RoboDK station: Estacion_feria_Con_Emergencia.rdk

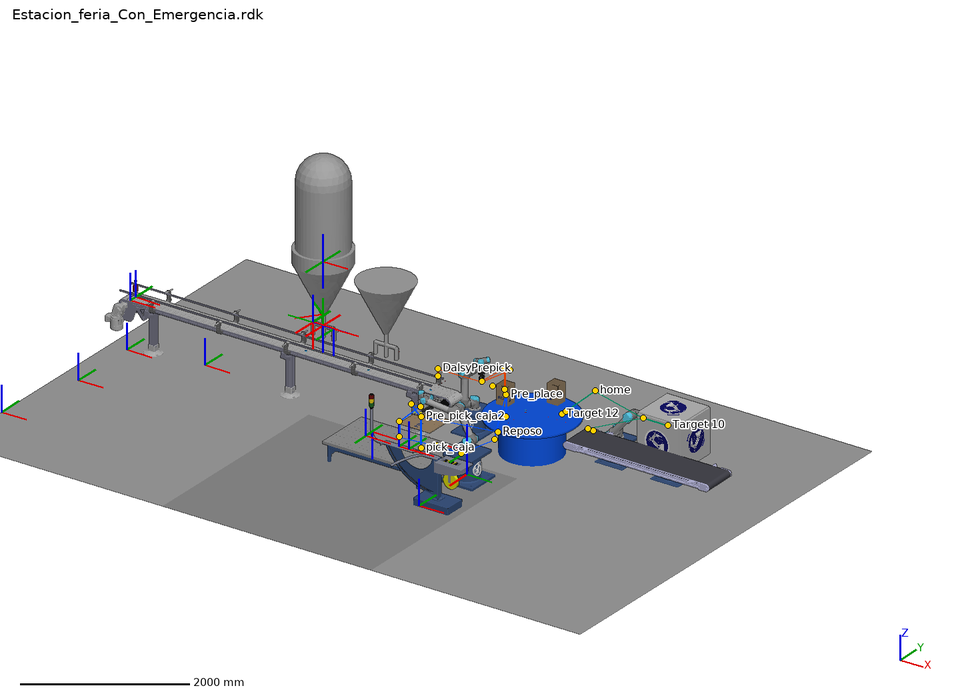
[picture v0: the station drawn from its stored meshes, robots at their saved joint values, targets as dots, program paths as lines]
Station EstacionProyectoFinaleliminarBotela (saved by RoboDK 5.9.4). Poses are relative to the parent item; angles as X-Y-Z fixed-axis rotations.
Station parameters (name, value as stored): Posicion, [[ 2850.000 ]] , CantBot1, 0, NUMBOTELLA1, 0, ElimBotellas1, 0, detectado1, 0, repes1, 0, Prellena1, 0, Prellena, 0, Detectado1, 0, IO_5, 1, NewPick, 0, Pinza, 1, NewPlace, 0, waituntil Detectado1, 1, Ventosa_plegado_caja, 1, CantCaja, 0.0, SCajaInicial, 0, SCajaPlace, 0, if(SCajaInicial, SyntaxError: Unexpected token `=', If(SCajaInicial, SyntaxError: Unexpected token `=', Mesa, 1, Mesa1, 0, Mesa2, 0, Mesa3, 1, MesaE, 1, MesaS, 1, Temperatura, 0, LotesPendientes, 1, SensorMqtt, 0, Ini_Detecta_Caja, 0, EMERGENCIA, 0
  - folder ESTACIÓN
    - folder Suelo
      - object Floor at (4500, 1500, 0) mm, size 3000 x 3000 x 0 mm, geometry from Floor.sld
      - object Floor2 at (1500, 1500, 0) mm, size 3000 x 3000 x 0 mm, geometry from Floor.sld
      - object Floor3 at (1500, 4500, 0) mm, size 3000 x 3000 x 0 mm, geometry from Floor.sld
      - object Floor4 at (4500, 4500, 0) mm, size 3000 x 3000 x 0 mm, geometry from Floor.sld
      - object Floor6 at (7500, 1500, 0) mm, size 3000 x 3000 x 0 mm, geometry from Floor.sld
      - object Floor5 at (7500, 4500, 0) mm, size 3000 x 3000 x 0 mm, geometry from Floor.sld
    - folder EMERGENCIA
      - program EMERGENCIA (3 instructions, listed below)
  - frame SisGeneral at (0, -19.13, 0) mm
    - folder SuministraCajas
      - frame SisCajas at (0, 1000, 0) mm
        - frame UR5 Base Cajas at (5520.28, 1665, 362.1) mm, rotated rx 0 ry 0 rz 180 deg
          - robot UR5 PrepCajas (model UR5): 6 axes
              modified DH rows (alpha deg, a mm, theta deg, d mm): 0, 0, 0, 89.2; 90, 0, 180, 0; 0, 425, 0, 0; 0, 392, 0, 109.3; -90, 0, 0, 94.75; 90, 0, 180, 82.5
              joint limits [-360, -360, -360, -360, -360, -360] to [360, 360, 360, 360, 360, 360]; home [0, -90, -90, 0, 90, 0]; saved at [7.72, -115.341, -54.372, -100.287, 90, 97.72]
            - frame Generic Box Erector Gripper Base at (0, 1000, 0) mm
            - robot Vplegadocaja: 1 axes
                modified DH rows (alpha deg, a mm, theta deg, d mm): 0, 0, 0, 0
                base shift (0, -125, 110) mm, rotated rx 0 ry 90 rz 0 deg
                joint limits [0] to [90]; home [0]; saved at [90]
              - tool Ventosa_plegado_caja, TCP at (0, 0, 200) mm
                - object Caja_plegada at (-6.06, -103.79, -200.38) mm, rotated rx 0 ry -90 rz 0 deg, size 213.4 x 213.4 x 444 mm, geometry from Box-215x215mm-Fold-2.sld
                - object caja_cintada at (15.94, -103.79, -200.38) mm, rotated rx 0 ry -90 rz 0 deg, size 160.1 x 160.1 x 259.7 mm, geometry from Box-215x215mm-Fold-3.sld
                - object Caja at (-171.32, 14.39, -556.39) mm, rotated rx 90 ry 0 rz 0 deg, size 444 x 419.7 x 11.5 mm, geometry from Box-215x215mm-Unfolded.sld
          - frame CoordBase_pedestal_caja at (-4.43, 0, -300) mm, rotated rx 0 ry 0 rz 90 deg
            - object Pedestal R1 at (0, 0, -60) mm, size 480 x 480 x 365.8 mm, geometry from Pedestal-H12in-Type-1.sld
          - target Reposo (Cartesian target) at (-498.67, 66.18, 420.87) mm, rotated rx 178.02 ry -0.17 rz 90 deg; joints [184.99, -90.98, -90.12, -90.89, 90, 4.99] of UR5 PrepCajas
          - target Pre_pick_caja2 (Cartesian target) at (671.03, -19.34, 260.81) mm, rotated rx 180 ry 0 rz 180 deg; joints [7.72, -117.384, -80.943, -71.673, 90, 97.72] of UR5 PrepCajas
          - target pick_caja (Cartesian target) at (671.03, -19.34, -150.19) mm, rotated rx 180 ry 0 rz 180 deg; joints [7.72, -132.159, -91.765, -46.076, 90, 97.72] of UR5 PrepCajas
          - target Giro (Cartesian target) at (580.93, 308.91, 583.09) mm, rotated rx 0 ry 90 rz 90 deg; joints [31.389, -172.181, 52.722, -60.541, 148.611, 90] of UR5 PrepCajas
          - target Paso_cintadora (Cartesian target) at (395, 385.89, 633.19) mm, rotated rx -45 ry 90 rz 45 deg; joints [50.203, -102.986, -71.875, -5.139, 129.797, 90] of UR5 PrepCajas
          - target Pre_abajo (Cartesian target) at (425, 775.89, 583.19) mm, rotated rx -45 ry 90 rz 45 deg; joints [58.921, -126.768, -44.607, -8.625, 121.079, 90] of UR5 PrepCajas
          - target abajo (Cartesian target) at (425, 775.89, 383.19) mm, rotated rx -45 ry 90 rz 45 deg; joints [58.921, -129.684, -69.347, 19.031, 121.079, 90] of UR5 PrepCajas
          - target fin_abajo (Cartesian target) at (-65, 715.89, 383.19) mm, rotated rx -45 ry 90 rz 45 deg; joints [112.972, -103.11, -110.097, 33.206, 67.028, 90] of UR5 PrepCajas
          - target cinta_abajo (Cartesian target) at (-425, 715.89, 383.19) mm, rotated rx -45 ry 90 rz 45 deg; joints [144.814, -123.817, -79.292, 23.109, 35.186, 90] of UR5 PrepCajas
          - target Paso_mesa (Cartesian target) at (-584.3, 268.15, 429.86) mm, rotated rx -90 ry 90 rz 90 deg; joints [162.957, -116.563, -83.461, 20.024, 107.043, 90] of UR5 PrepCajas
          - target Pre_place (Cartesian target) at (-128.1, -624.3, 529.86) mm, rotated rx 45 ry 90 rz -45 deg; joints [266.879, -85.143, -106.269, 11.412, 93.122, 90] of UR5 PrepCajas
          - target Place (Cartesian target) at (-128.1, -624.3, 241.86) mm, rotated rx 45 ry 90 rz -45 deg; joints [266.879, -110.903, -128.99, 59.893, 93.122, 90] of UR5 PrepCajas
        - frame Mesa at (4197.94, 1472.94, 273.52) mm
          - object mesa_caja at (0, 0, 0) mm, size 1420 x 820 x 800 mm, geometry from Table-1400x800x800mm.sld
          - frame Mesa_caja at (480, 0, 0) mm
          - object Sensor_caja_inicial at (650, -170, 0) mm, rotated rx 0 ry 0 rz 90 deg, size 683.3 x 45.2 x 12.5 mm, geometry from SICK-WL4S-Laser-Sensor.sld
        - frame Sistema_plegadora at (5470, 760, 0) mm
          - frame Caja_plegadora at (-210, 90, 650) mm
          - object Box Erector Station at (180, 120, 0) mm, rotated rx 0 ry 0 rz -90 deg, size 477.6 x 1402.8 x 1195.5 mm, geometry from Box-Erector-Station.sld
      - folder Programas_RDK
        - program Pick_place_caja (41 instructions, listed below)
        - program Main_sensor (11 instructions, listed below)
      - folder Programas_python
        - Python program ResetCaja (listed below)
        - Python program 2_caja (listed below)
        - Python program 3_caja (listed below)
        - Python program Abrir_Herramienta (listed below)
        - Python program Cerrar_heramienta (listed below)
        - Python program Copiar_caja_place (listed below)
        - Python program Inicializar_contador (listed below)
        - Python program Sensor_inicial (listed below)
        - Python program Sensor_place (listed below)
        - Python program QuitarCajasOcultas (listed below)
    - folder CintayRobot
      - frame SisRefPick at (250, 2217.22, 0) mm
        - frame Cinta Botellas 1 at (0, 1000, 0) mm
          - robot CintaUno: 1 axes
              modified DH rows (alpha deg, a mm, theta deg, d mm): 0, 0, 0, 0 linear
              base shift (0, 0, 0) mm, rotated rx 0 ry 90 rz 0 deg
              joint limits [0] to [4500]; home [0]; saved at [50]
            - frame FrameBotellaSave at (0, 0, 0) mm
              - object Guardado at (0, 0, 0) mm, size 71.4 x 71.4 x 225.2 mm, geometry from Bottle-Label.sld
            - frame Move at (0, 0, 0) mm
              - frame FrameBotella at (0, 100, 0) mm
                - object Guardado at (0, 0, 0) mm, size 71.4 x 71.4 x 225.2 mm, geometry from Bottle-Label.sld
                - object botella0.0 at (0, 0, 0) mm, size 71.4 x 71.4 x 225.2 mm, geometry from Bottle-Label.sld
          - target Inicio (Cartesian target) at (0, 100, 863) mm; joints [0] of CintaUno
          - target Final (Cartesian target) at (4325.5, 559.3, 913.95) mm, rotated rx -90 ry 0 rz 90 deg; joints [0, -90, -90, 0, 90, 0] of CintaUno
          - frame TANQUE 1 at (1750, -902.14, 647.6) mm
            - frame Cono at (1000, 1000, 1240) mm, rotated rx 180 ry 0 rz 0 deg
              - object Cone 500x500mm at (0, 0, 0) mm, size 746.2 x 750 x 750 mm, geometry from Cone-500x500mm.sld
            - frame Deposito at (1000, 1000, 1240) mm
              - object Deposito at (0, 0, 0) mm, size 750 x 750 x 1389.5 mm, geometry from Light-Off.sld
            - frame Frame 24 at (1000.71, 1000.6, 551.36) mm, rotated rx 180 ry 0 rz -124.91 deg
              - object Cylinder 50x150mm at (0, 0, 0) mm, size 50 x 50 x 150 mm, geometry from Cylinder-50x150mm.sld
            - frame Frame 25 at (1000.71, 1000.6, 401.36) mm, rotated rx -180 ry 0 rz -90 deg
              - object Cylinder 50x150mm at (0, 0, 0) mm, size 50 x 50 x 150 mm, geometry from Cylinder-50x150mm.sld
            - frame Frame 26 at (1000.71, 1000.6, 401.36) mm, rotated rx 90 ry 0 rz 90 deg
              - object Cylinder 50x150mm at (0, 0, 0) mm, size 50 x 50 x 150 mm, geometry from Cylinder-50x150mm.sld
            - frame Frame 27 at (1150.71, 1000.6, 401.36) mm, rotated rx -180 ry 0 rz 0 deg
              - object Cylinder 50x150mm at (0, 0, 0) mm, size 50 x 50 x 150 mm, geometry from Cylinder-50x150mm.sld
            - frame Frame 25 at (1000.71, 1000.6, 401.36) mm, rotated rx -180 ry 0 rz -90 deg
              - object Cylinder 50x150mm at (0, 0, 0) mm, size 50 x 50 x 150 mm, geometry from Cylinder-50x150mm.sld
            - frame Frame 25 at (850.71, 1000.6, 401.36) mm, rotated rx -180 ry 0 rz -90 deg
              - object Cylinder 50x150mm at (0, 0, 0) mm, size 50 x 50 x 150 mm, geometry from Cylinder-50x150mm.sld
            - frame Frame 25 at (850.71, 1000.6, 401.36) mm, rotated rx 0 ry 90 rz 0 deg
              - object Cylinder 50x150mm at (0, 0, 0) mm, size 50 x 50 x 150 mm, geometry from Cylinder-50x150mm.sld
            - frame Frame 31 at (850.65, 1001.38, 406.13) mm
              - object Sphere D100mm at (0, 0, 0) mm, size 50 x 50 x 50 mm, geometry from Sphere-D100mm.sld
            - frame Frame 31 at (1151.57, 999.51, 402.52) mm
              - object Sphere D100mm at (0, 0, 0) mm, size 50 x 50 x 50 mm, geometry from Sphere-D100mm.sld
          - frame DispensaTapones at (2650, -902.14, 647.6) mm
            - frame Cono at (1000, 1000, 1240) mm, rotated rx 180 ry 0 rz 0 deg
              - object Cone 500x500mm at (0, 0, 0) mm, size 746.2 x 750 x 750 mm, geometry from Cone-500x500mm.sld
            - frame Frame 24 at (1000.71, 1000.6, 551.36) mm, rotated rx 180 ry 0 rz -124.91 deg
              - object Cylinder 50x150mm at (0, 0, 0) mm, size 50 x 50 x 150 mm, geometry from Cylinder-50x150mm.sld
            - frame Frame 25 at (1000.71, 1000.6, 401.36) mm, rotated rx -180 ry 0 rz -90 deg
              - object Cylinder 50x150mm at (0, 0, 0) mm, size 50 x 50 x 150 mm, geometry from Cylinder-50x150mm.sld
            - frame Frame 26 at (1000.71, 1000.6, 401.36) mm, rotated rx 90 ry 0 rz 90 deg
              - object Cylinder 50x150mm at (0, 0, 0) mm, size 50 x 50 x 150 mm, geometry from Cylinder-50x150mm.sld
            - frame Frame 27 at (1150.71, 1000.6, 401.36) mm, rotated rx -180 ry 0 rz 0 deg
              - object Cylinder 50x150mm at (0, 0, 0) mm, size 50 x 50 x 150 mm, geometry from Cylinder-50x150mm.sld
            - frame Frame 25 at (1000.71, 1000.6, 401.36) mm, rotated rx -180 ry 0 rz -90 deg
              - object Cylinder 50x150mm at (0, 0, 0) mm, size 50 x 50 x 150 mm, geometry from Cylinder-50x150mm.sld
            - frame Frame 25 at (850.71, 1000.6, 401.36) mm, rotated rx -180 ry 0 rz -90 deg
              - object Cylinder 50x150mm at (0, 0, 0) mm, size 50 x 50 x 150 mm, geometry from Cylinder-50x150mm.sld
            - frame Frame 25 at (850.71, 1000.6, 401.36) mm, rotated rx 0 ry 90 rz 0 deg
              - object Cylinder 50x150mm at (0, 0, 0) mm, size 50 x 50 x 150 mm, geometry from Cylinder-50x150mm.sld
            - frame Frame 31 at (850.65, 1001.38, 406.13) mm
              - object Sphere D100mm at (0, 0, 0) mm, size 50 x 50 x 50 mm, geometry from Sphere-D100mm.sld
            - frame Frame 31 at (1151.57, 999.51, 402.52) mm
              - object Sphere D100mm at (0, 0, 0) mm, size 50 x 50 x 50 mm, geometry from Sphere-D100mm.sld
          - frame Sensor3 at (3498.8, -14.22, 715.35) mm, rotated rx 0 ry 0 rz 88.62 deg
            - object B2 at (0, 0, 0) mm, size 683.3 x 45.2 x 12.5 mm, geometry from SICK-WL4S-Laser-Sensor.sld
          - frame Sensor2 at (4402.28, -29.98, 715.35) mm, rotated rx 0 ry 0 rz 88.62 deg
            - object B1 at (0, 0, 0) mm, size 683.3 x 45.2 x 12.5 mm, geometry from SICK-WL4S-Laser-Sensor.sld
          - frame Sensor1 at (2598.8, -14.22, 715.35) mm, rotated rx 0 ry 0 rz 88.62 deg
            - object B0 at (0, 0, 0) mm, size 683.3 x 45.2 x 12.5 mm, geometry from SICK-WL4S-Laser-Sensor.sld
          - target DalsyPrepick (Cartesian target) at (4404.64, 97.25, 945.23) mm, rotated rx -179.46 ry -0.56 rz 92.6 deg; joints [67.794, -102.103, -28.32, -139.861, 89.279, 65.196] of UR5PickDalsy
          - target DalsyPick (Cartesian target) at (4400.29, 94.49, 846.14) mm, rotated rx -179.46 ry -0.56 rz 92.6 deg; joints [67.407, -90.716, -60.305, -119.258, 89.278, 64.809] of UR5PickDalsy
          - target DalsyPuntoPaso (Cartesian target) at (4989.54, 154.84, 921.17) mm, rotated rx 176.54 ry 3.78 rz 107.72 deg; joints [150.48, -91.95, -47.39, -125.54, 89.98, 132.65] of UR5PickDalsy
          - target PuntoDePaso2 (Cartesian target) at (5091.93, 592.06, 921.34) mm, rotated rx 176.53 ry 3.81 rz 169.24 deg; joints [212.01, -91.94, -47.38, -125.53, 89.97, 132.65] of UR5PickDalsy
          - target PrePlace (Cartesian target) at (5051.88, 544.46, 950.34) mm, rotated rx 179.87 ry 0 rz -95.46 deg; joints [208.979, -92.535, -38.825, -138.744, 90.075, 34.439] of UR5PickDalsy
          - target DalsyPlace (Cartesian target) at (5051.88, 544.46, 680.34) mm, rotated rx 179.87 ry 0 rz -95.46 deg; joints [208.979, -74.687, -99.618, -95.799, 90.075, 34.439] of UR5PickDalsy
          - target Target 9 (Cartesian target) at (5079.28, 251.73, 846.24) mm, rotated rx -179.45 ry -0.55 rz -167.69 deg; joints [167.11, -90.71, -60.3, -119.25, 89.27, 64.8] of UR5PickDalsy
          - target Target 10 (Cartesian target) at (7103.35, 957.35, 614.14) mm, rotated rx -138.15 ry 89.07 rz -48.26 deg; joints [177.195, -131.024, -49.86, -164.778, 177.217, -76.295] of UR5 SalidaCjas
          - target Target 11 (Cartesian target) at (4404.64, 97.25, 945.23) mm, rotated rx -179.46 ry -0.56 rz 92.6 deg; joints [67.794, -102.103, -28.32, -139.861, 89.279, 65.196] of UR5PickDalsy
          - target Target 12 (Cartesian target) at (5875.13, 535.29, 591.77) mm, rotated rx -124.69 ry 88.93 rz 144.57 deg; joints [23.154, -118.729, -72.709, -170.068, 203.904, -92.258] of UR5 SalidaCjas
        - frame UR5 BasePickDalsy at (4673.46, 1459.5, 355) mm, rotated rx 0 ry 0 rz 180 deg
          - robot UR5PickDalsy (model UR5): 6 axes
              modified DH rows (alpha deg, a mm, theta deg, d mm): 0, 0, 0, 89.2; 90, 0, 180, 0; 0, 425, 0, 0; 0, 392, 0, 109.3; -90, 0, 0, 94.75; 90, 0, 180, 82.5
              joint limits [-360, -360, -360, -360, -360, -360] to [360, 360, 360, 360, 360, 360]; home [0, -90, -90, 0, 90, 0]; saved at [150.48, -91.95, -47.39, -125.54, 89.98, 132.65]
            - tool GripperPick, TCP at (0, 0, 130) mm, size 147.4 x 75 x 146.8 mm
            - tool GripperPickV, TCP at (0, 0, 130) mm, size 134.4 x 75 x 157.6 mm
          - frame Frame 45 at (4.13, 0, -300) mm
            - object Pedestal R1 at (0, 0, 0) mm, size 400 x 400 x 304.8 mm, geometry from Pedestal-H12in-Type-1.sld
      - folder ProgramasDeLaCinta
        - Python program AvanzaCinta1 (listed below)
        - Python program AvanzaCinta2 (listed below)
        - Python program ResetBot (listed below)
        - program ProgCinta1 (15 instructions, listed below)
        - Python program ProgCintaUno (listed below)
      - folder Sensores
        - Python program ProgB0 (listed below)
        - Python program ProgB1 (listed below)
        - Python program ProgB2 (listed below)
      - folder ProgramasUr
        - program DalsyPickPlace (33 instructions, listed below)
        - Python program PickDalsy (listed below)
        - Python program PlaceDalsy (listed below)
        - Python program BorrarBotella (listed below)
        - Python program RobotPickAndPlace (listed below)
    - folder CerradoCajas
      - frame SisSalida at (6887.77, 2000, 0) mm
        - frame UR5BaseSalidaCajas at (-200.53, 2100.2, 305) mm, rotated rx 0 ry 0 rz 180 deg
          - robot UR5 SalidaCjas (model UR5): 6 axes
              modified DH rows (alpha deg, a mm, theta deg, d mm): 0, 0, 0, 89.2; 90, 0, 180, 0; 0, 425, 0, 0; 0, 392, 0, 109.3; -90, 0, 0, 94.75; 90, 0, 180, 82.5
              joint limits [-360, -360, -360, -360, -360, -360] to [360, 360, 360, 360, 360, 360]; home [0, -90, -90, 0, 90, 0]; saved at [177.195, -131.024, -49.86, -164.778, 177.217, -76.295]
            - tool VentosaSalida, TCP at (0, 22.5, 135) mm, size 179.2 x 110.2 x 138.7 mm
              - object caja_cerradaPLANTILLA at (2.18, 97.23, 6.23) mm, rotated rx 90.61 ry -0.74 rz -89.13 deg, size 160.1 x 160.1 x 186.3 mm, geometry from Box-215x215mm-Folded(2).sld
          - frame CoordBase at (0, 0, -320) mm, rotated rx -0.35 ry 0 rz 0 deg
            - object Pedestal R1 at (0, 0, 0) mm, size 400 x 400 x 304.8 mm, geometry from Pedestal-H12in-Type-1.sld
          - target pick_cajamesa (Cartesian target) at (562.11, 347.69, 286.77) mm, rotated rx -124.69 ry 88.93 rz -35.43 deg; joints [23.154, -118.729, -72.709, -170.068, 203.904, -92.258] of UR5 SalidaCjas
          - target prepick_cajamesa (Cartesian target) at (561.01, 262.7, 287.67) mm, rotated rx -124.69 ry 88.93 rz -35.43 deg; joints [15.242, -116.952, -75.276, -169.987, 195.996, -93.011] of UR5 SalidaCjas
          - target home (Cartesian target) at (209.75, 166.03, 613.52) mm, rotated rx -26.26 ry 79.18 rz 65.79 deg; joints [15.24, -64.23, -88.13, -169.98, 195.99, -58.26] of UR5 SalidaCjas
          - frame SisCubo at (-800, 0, -320) mm, rotated rx -0.35 ry 0 rz 0 deg
            - object Pedestal R1 at (0, 0, 0) mm, size 400 x 400 x 304.8 mm, geometry from Pedestal-H12in-Type-1.sld
            - object Cubo at (-300, -300, 300) mm, rotated rx 90 ry 0 rz 0 deg, size 636 x 636 x 672 mm
          - target pre_cajacubo (Cartesian target) at (-316.13, -74.99, 305.37) mm, rotated rx -138.15 ry 89.07 rz 131.74 deg; joints [174.473, -84.902, -111.44, -156.399, 174.538, -83.391] of UR5 SalidaCjas
          - target dentro_cajacubo (Cartesian target) at (-666.11, -74.37, 309.14) mm, rotated rx -138.15 ry 89.07 rz 131.74 deg; joints [177.195, -131.024, -49.86, -164.778, 177.217, -76.295] of UR5 SalidaCjas
          - target place_cajacinta (Cartesian target) at (-20.88, 535.48, 307.78) mm, rotated rx -142.74 ry 89.07 rz 36.86 deg; joints [81.199, -115.849, -73.914, 194.832, 171.57, 274.45] of UR5 SalidaCjas
          - target preplace_cajacinta (Cartesian target) at (54.12, 534.95, 308.76) mm, rotated rx -142.74 ry 89.07 rz 36.86 deg; joints [74.123, -120.474, -66.715, 189.969, 164.509, 272.115] of UR5 SalidaCjas
        - frame cinta2 at (-383.81, 1308.32, 516.62) mm, rotated rx 0.97 ry 0 rz 0 deg
          - robot CintaSalidas: 1 axes
              modified DH rows (alpha deg, a mm, theta deg, d mm): 0, 0, 0, 0 linear
              base shift (0, 0, 0) mm, rotated rx 0 ry 90 rz 0 deg
              joint limits [-500000] to [500000]; home [0]; saved at [-500000]
      - folder scripts
        - program Prog_cajasSalida (23 instructions, listed below)
        - folder pyt
          - Python program SensorDetectaCaja (listed below)
          - Python program Plantilla (listed below)
          - Python program AvanzaCajasSalida (listed below)
        - folder rdk
    - folder Mesa
      - frame MesaGiratoriaBase at (5724.13, 3717.02, 0) mm
        - robot MesaGiratoria: 1 axes
            modified DH rows (alpha deg, a mm, theta deg, d mm): 0, 0, 0, 0
            joint limits [-200] to [200]; home [0]; saved at [110]
          - frame SistMesaGiratoria at (0, 1000, 0) mm
          - frame Place_caja at (-410, 300, 573) mm, rotated rx 0 ry 0 rz -40 deg
            - object cajaplace1.0 at (310.2, 492.2, 15.02) mm, rotated rx 0 ry 0 rz -70 deg, size 160.1 x 160.1 x 259.7 mm, geometry from Box-215x215mm-Fold-3.sld
            - object cajaplace0.0 at (965.38, 230.44, 15.02) mm, rotated rx 0 ry 0 rz -160 deg, size 160.1 x 160.1 x 259.7 mm, geometry from Box-215x215mm-Fold-3.sld
        - folder ScriptsMesa
          - Python program MoverMesa (listed below)
          - program MoverMesaBucle (8 instructions, listed below)
        - object Sensor_place_caja at (-90, -30, 510) mm, rotated rx 0 ry 0 rz -90 deg, size 683.3 x 45.2 x 12.5 mm, geometry from SICK-WL4S-Laser-Sensor.sld
        - object SensorDetectaCajaSalida at (-100, -10, 510) mm, size 683.3 x 45.2 x 12.5 mm, geometry from SICK-WL4S-Laser-Sensor.sld
  - folder PROGRAMA_PRINCIPAL
    - program Main (17 instructions, listed below)
  - folder MQTT
    - Python program mqttlistenerCinta (listed below)
    - Python program RobotControllerCinta (listed below)
    - Python program mqttlistenerTEMP (listed below)
    - Python program mqttlistenerDecCaja (listed below)
    - Python program RobotControllerTEMP (listed below)
    - Python program RobotControllerDecCaja (listed below)
  - folder Basedatos
    - folder BaseDeDatos
      - Python program ConsultarBD (listed below)
      - Python program CrearBotellaBD (listed below)
      - Python program LlenarBD (listed below)
      - Python program ResetBD (listed below)
      - Python program EmpaquetarBD (listed below)
      - Python program TaponarBD (listed below)
    - folder JugarBD
      - Python program CrearLotesBD (listed below)
      - Python program TerminarLotesBD (listed below)
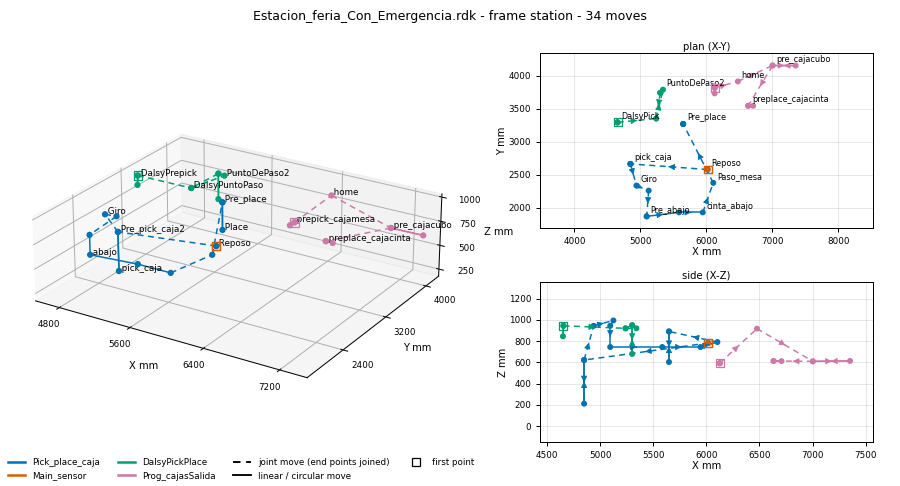
[picture p0: tool path of Estacion_feria_Con_Emergencia.rdk in frame station, 34 of 34 moves have a stored position in this frame; points joined in program order, loops and branches not executed]

--- program EMERGENCIA (robot UR5 PrepCajas) ---
  while EMERGENCIA ==1
  Pausa 500 ms
  end

--- program Pick_place_caja (robot UR5 PrepCajas) ---
  Est. Ref.: UR5 Base Cajas
  Est. herr: Ventosa_plegado_caja
  Establecer velocidad (500.0 mm/s)
  while Mesa==0
  Pausa 500 ms
  end
  Mesa=0
  MoveJ (Reposo)
  Llamar Abrir_Herramienta
  MoveJ (Pre_pick_caja2)
  Establecer velocidad (40.0 mm/s)
  MoveL (pick_caja)
  Set Ventosa_plegado_caja=1
  Adjuntar a Ventosa_plegado_caja
  Pausa 500 ms
  MoveL (Pre_pick_caja) -> target Pre_pick_caja2
  Establecer velocidad (500.0 mm/s)
  Llamar Cerrar_heramienta
  Llamar 2_caja
  Pausa 500 ms
  MoveJ (Giro)
  MoveJ (Paso_cintadora)
  MoveJ (Pre_abajo)
  Establecer velocidad (100.0 mm/s)
  MoveL (abajo)
  MoveL (fin_abajo)
  Llamar 3_caja
  MoveL (cinta_abajo)
  Establecer velocidad (500.0 mm/s)
  MoveJ (Paso_mesa)
  MoveJ (Pre_place)
  Establecer velocidad (100.0 mm/s)
  MoveL (Place)
  Set Ventosa_plegado_caja=0
  Separar de Ventosa_plegado_caja
  Pausa 500 ms
  Llamar Copiar_caja_place
  MoveL (Pre_place)
  Llamar ResetCaja
  Llamar QuitarCajasOcultas
  Mesa2=1

--- program Main_sensor (robot UR5 PrepCajas) ---
  Est. herr: Ventosa_plegado_caja
  Est. Ref.: UR5 Base Cajas
  MoveJ (Reposo)
  IF SCajaInicial == 1 THEN
  IF SCajaPlace==0 Then
  while Ini_Detecta_Caja == 0
  Pausa 500 ms
  end
  Llamar Pick_place_caja
  ENDIF
  ENDIF

--- Python program ResetCaja ---
from robodk import robolink
from robodk import robomath

# Conexión con RoboDK
RDK = robolink.Robolink()

# -------- OBTENER OBJETOS --------
caja = RDK.Item('Caja', robolink.ITEM_TYPE_OBJECT)
mesa_caja = RDK.Item('Mesa_caja', robolink.ITEM_TYPE_FRAME)

# -------- COMPROBACIONES --------
if not caja.Valid():
    raise Exception("No se encontró el objeto 'Caja'")

if not mesa_caja.Valid():
    raise Exception("No se encontró el sistema de coordenadas 'Mesa_caja'")

# -------- REINICIAR CAJA INICIAL --------

# Hacer que la caja dependa del frame Mesa_caja
caja.setParentStatic(mesa_caja)

# Definir la pose [x,y,z,rx,ry,rz] = [0,0,0,0,0,0] PARA PONERLO EN LA MESA
pose_origen = robomath.xyzrpw_2_pose([0, 0, 0, 0, 0, 0])

# Aplicar la pose a la caja
caja.setPose(pose_origen)

caja.setVisible(True,True)  #PONGO VISIBLE LA CAJA
RDK.Render()

#QUITO LAS CAJAS LAS CUALES USO PARA LA ANIMACION
caja2 = RDK.Item('Caja_plegada')
if not caja2.Valid():
    raise Exception('No se encontró el objeto Caja_plegada')

caja2.setVisible(False,False)
RDK.Render()

caja3=RDK.Item('Caja_cintada')
if not caja3.Valid():
    raise Exception('NO hay caja')

caja3.setVisible(False,False)
RDK.Render()

--- Python program 2_caja ---
# Type help("robodk.robolink") or help("robodk.robomath") for more information
# Press F5 to run the script
# Documentation: https://robodk.com/doc/en/RoboDK-API.html
# Reference:     https://robodk.com/doc/en/PythonAPI/robodk.html
# Note: It is not required to keep a copy of this file, your Python script is saved with your RDK project

# You can also use the new version of the API:
from robodk import robolink    # RoboDK API
from robodk import robomath    # Robot toolbox
RDK = robolink.Robolink()

from robodk.robolink import *
from robodk.robomath import *

#CODIGO DE LA CAJA SIN HACER NINGUNA MODIFICACION

cajainicial=RDK.Item('Caja') #CREO LA CAJA
if not cajainicial.Valid(): #COMPRUEBO QUE EXISTA LA CAJA
    raise Exception('Caja inicial no encontrada') #SINO LANZO UNA EXCEPCIONN

#------------------------------------------------
# CODIGGO PARA PONER CAJA '2ºESTADO' EN LA HERRAMIENTA

#HERRAMIENTA
tool = RDK.Item('Ventosa_plegado_caja', ITEM_TYPE_TOOL)#CREO ITEM HERRAMIENTA
if not tool.Valid(): #COMPRUEBO QUE EXISTA LA VENTOSA
    raise Exception('No se encontró la herramienta Ventosa_plegado_caja')#SINO LANZO UNA EXCEPCIONN
#----------------------------------------------------

#CAJA 2ºESTADO
caja = RDK.Item('Caja_plegada') #CREO LA CAJA EN SU 2ºESTADO
if not caja.Valid(): #COMPRUEBO QUE EXISTA ESA CAJA
    raise Exception('No se encontró el objeto Caja_plegada') #SINO LANZO UNA EXCEPCIONN

#----------------------------------------------------
# Hacer visible la caja
cajainicial.setVisible(False,False) #1.PONGO LA CAJA INICIAL INVISIBLE


#VOY A INSERTAR LA CAJA EN SU 2º ESTDO DENTRO DEL SISTEMA DE REFERENCIA DE LA VENTOSA
#ES DECIR PONDRE LA CAJA EN LA HERRAMIENTA POR CODIGO.
caja.setParentStatic(tool)

#VARIABLE POSE DONDE IRA LA CAJA
pose_herramienta = xyzrpw_2_pose([-6.063, -103.794, -200.377, 0, -90, 0])

# Aplicar la pose a la caja
caja.setPose(pose_herramienta)
# Hacer visible la caja
cajainicial.setVisible(False,False) #1.PONGO LA CAJA INICIAL INVISIBLE

caja.setVisible(True, True)

RDK.Render()

--- Python program 3_caja ---
# Type help("robodk.robolink") or help("robodk.robomath") for more information
# Press F5 to run the script
# Documentation: https://robodk.com/doc/en/RoboDK-API.html
# Reference:     https://robodk.com/doc/en/PythonAPI/robodk.html
# Note: It is not required to keep a copy of this file, your Python script is saved with your RDK project

# You can also use the new version of the API:
from robodk import robolink    # RoboDK API
from robodk import robomath    # Robot toolbox
RDK = robolink.Robolink()

from robodk.robolink import *
from robodk.robomath import *
#Fragmento de codigo donde hacemos invisible la caja sin cerrar la parte inferiro
caja=RDK.Item('Caja_plegada')
if not caja.Valid():
    raise Exception('No se encontro el objeto caja_plegada')

caja.setVisible(False,False)
RDK.Render()

#Fragmento de codigo donde hacemos invisible la caja con la parte inferior plegada
caja_abajo=RDK.Item('Caja_cintada')
tool=RDK.Item('Ventosa_plegado_caja', ITEM_TYPE_TOOL)
if not(caja_abajo.Valid()):
    raise Exception('Caja_cintada no se ha encontrado')
if not(tool.Valid()):
    raise Exception('No se ha conseguido unir a la ventosa')

caja_abajo.setVisible(True, True)
#Meter ne el sistema de referencia de la herramienta
caja_abajo.setParentStatic(tool)

pose_ventosa=xyzrpw_2_pose([15.937 , -103.794, -200.377, 0.00, -90.00, 0.00])
caja_abajo.setPose(pose_ventosa)
RDK.Render()

--- Python program Abrir_Herramienta ---
# Type help("robodk.robolink") or help("robodk.robomath") for more information
# Press F5 to run the script
# Documentation: https://robodk.com/doc/en/RoboDK-API.html
# Reference:     https://robodk.com/doc/en/PythonAPI/robodk.html
# Note: It is not required to keep a copy of this file, your Python script is saved with your RDK project

# You can also use the new version of the API:
from robodk import robolink    # RoboDK API
from robodk import robomath    # Robot toolbox

from robodk.robolink import Robolink

# Conectar con RoboDK
RDK = Robolink()

# Obtener la herramienta (mecanismo)
tool = RDK.Item('Vplegadocaja')

if not tool.Valid():
    raise Exception('No se encontró la herramienta Vplegadocaja')

# Obtener joints actuales de la herramienta
joints = tool.Joints().list()

if len(joints) == 0:
    raise Exception('La herramienta no tiene ejes articulares')

# Sumar 75 grados al eje deseado (J1 = índice 0)
joints[0] = joints[0] + 90

# Aplicar el pilotaje articular
tool.setJoints(joints)

--- Python program Cerrar_heramienta ---
# Type help("robodk.robolink") or help("robodk.robomath") for more information
# Press F5 to run the script
# Documentation: https://robodk.com/doc/en/RoboDK-API.html
# Reference:     https://robodk.com/doc/en/PythonAPI/robodk.html
# Note: It is not required to keep a copy of this file, your Python script is saved with your RDK project

# You can also use the new version of the API:
from robodk import robolink    # RoboDK API
from robodk import robomath    # Robot toolbox
RDK = robolink.Robolink()

from robodk.robolink import Robolink

import time

# Conectar con RoboDK
RDK = Robolink()

# Obtener la herramienta (mecanismo)
tool = RDK.Item('Vplegadocaja')

if not tool.Valid():
    raise Exception('No se encontró la herramienta Vplegadocaja')

# Obtener joints actuales de la herramienta
joints = tool.Joints().list()

if len(joints) == 0:
    raise Exception('La herramienta no tiene ejes articulares')

# Sumar 75 grados al eje deseado (J1 = índice 0)
joints[0] = joints[0] -90

# Aplicar el pilotaje articular
tool.setJoints(joints)


time.sleep(0.02)

--- Python program Copiar_caja_place ---
# Type help("robodk.robolink") or help("robodk.robomath") for more information
# Press F5 to run the script
# Documentation: https://robodk.com/doc/en/RoboDK-API.html
# Reference:     https://robodk.com/doc/en/PythonAPI/robodk.html
# Note: It is not required to keep a copy of this file, your Python script is saved with your RDK project

# You can also use the new version of the API:
from robodk import robolink    # RoboDK API
from robodk import robomath    # Robot toolbox
RDK = robolink.Robolink()

caja=RDK.Item('caja_cintada')
SisMesa=RDK.Item('Place_caja')
CantCajas=RDK.getParam('CantCaja')

CantCajas=1+CantCajas
caja.Copy()
nueva_caja=RDK.Paste(SisMesa)
nueva_caja.setName(f'cajaplace{CantCajas}')

nueva_caja.setVisible(True, True)
RDK.Render()
caja.setVisible(False,False)
RDK.Render()


RDK.setParam('CantCaja',CantCajas)

--- Python program Inicializar_contador ---
# Type help("robodk.robolink") or help("robodk.robomath") for more information
# Press F5 to run the script
# Documentation: https://robodk.com/doc/en/RoboDK-API.html
# Reference:     https://robodk.com/doc/en/PythonAPI/robodk.html
# Note: It is not required to keep a copy of this file, your Python script is saved with your RDK project

# You can also use the new version of the API:
from robodk import robolink    # RoboDK API
from robodk import robomath    # Robot toolbox
RDK = robolink.Robolink()

# Forward and backwards compatible use of the RoboDK API:
# Remove these 2 lines to follow python programming guidelines
from robodk import *      # RoboDK API
from robolink import *    # Robot toolbox


numCajas=RDK.getParam('CantCaja')
numCajas=0.0
RDK.setParam('CantCaja',numCajas)

--- Python program Sensor_inicial ---
# Type help("robodk.robolink") or help("robodk.robomath") for more information
# Press F5 to run the script
# Documentation: https://robodk.com/doc/en/RoboDK-API.html
# Reference:     https://robodk.com/doc/en/PythonAPI/robodk.html
# Note: It is not required to keep a copy of this file, your Python script is saved with your RDK project

# You can also use the new version of the API:
from robodk import robolink    # RoboDK API
from robodk import robomath    # Robot toolbox
RDK = robolink.Robolink()

#FRAGMENTO DE CODIGO DONDE MIRA SI HAY UNA CAJA INCIALMENTE
sensor=RDK.Item('Sensor_caja_inicial')
estado_detectado=0
caja=RDK.Item('Caja')



while True:

        if sensor.Collision(caja):
            estado_detectado=1
            RDK.setParam('SCajaInicial',estado_detectado)

        else:
            estado_detectado=0
            RDK.setParam('SCajaInicial',estado_detectado)
#.---------------------------FIN---------------------------

--- Python program Sensor_place ---
from robodk.robolink import Robolink
import time

RDK = Robolink()

sensor_mesa_giratoria = RDK.Item('Sensor_place_caja')

inicio = 1
estado_detectado = 0
cuenta = 0

caja = RDK.Item(f'cajaplace{inicio}.0')

while True:

    try:
        # Validar sensor
        if not sensor_mesa_giratoria.Valid():
            print("Sensor no válido")
            time.sleep(0.1)
            continue

        # Validar caja
        if not caja.Valid():
            inicio += 1
            caja = RDK.Item(f'cajaplace{inicio}.0')
            continue

        # 🔥 PROTEGER Collision
        try:
            detectado = 1 if sensor_mesa_giratoria.Collision(caja) else 0
        except:
            print("⚠ Timeout o error en Collision()")
            time.sleep(0.1)
            continue

        if detectado != estado_detectado:

            if detectado == 1:
                print(f"Caja {inicio} detectada")
                RDK.setParam('SCajaPlace', '1')
                cuenta += 1

            else:
                print(f"Caja {inicio} ha salido")
                RDK.setParam('SCajaPlace', '0')

                inicio += 1
                caja = RDK.Item(f'cajaplace{inicio}.0')

            estado_detectado = detectado

    except Exception as e:
        print("Error general:", e)

    # ⏱️ IMPORTANTE: bajar frecuencia
    time.sleep(0.05)

--- Python program QuitarCajasOcultas ---
# Type help("robodk.robolink") or help("robodk.robomath") for more information
# Press F5 to run the script
# Documentation: https://robodk.com/doc/en/RoboDK-API.html
# Reference:     https://robodk.com/doc/en/PythonAPI/robodk.html
# Note: It is not required to keep a copy of this file, your Python script is saved with your RDK project

# You can also use the new version of the API:
from robodk import robolink    # RoboDK API
from robodk import robomath    # Robot toolbox
RDK = robolink.Robolink()

# Forward and backwards compatible use of the RoboDK API:
# Remove these 2 lines to follow python programming guidelines
from robodk import *      # RoboDK API
from robolink import *    # Robot toolbox
# Link to RoboDK
# RDK = Robolink()

# Notify user:


tool = RDK.Item('Ventosa_plegado_caja')#CREO ITEM HERRAMIENTA


cajaplegada=RDK.Item('Caja_plegada')
caja_abajo=RDK.Item('Caja_cintada')


cajaplegada.setParentStatic(tool)
caja_abajo.setParentStatic(tool)

#VARIABLE POSE DONDE IRA LA CAJA
pose_herramienta = xyzrpw_2_pose([-6.063, -103.794, -200.377, 0, -90, 0])
pose_ventosa=xyzrpw_2_pose([15.937 , -103.794, -200.377, 0.00, -90.00, 0.00])

cajaplegada.setPose(pose_herramienta)
caja_abajo.setPose(pose_ventosa)


RDK.Render()

--- Python program AvanzaCinta1 ---
# Type help("robodk.robolink") or help("robodk.robomath") for more information
# Press F5 to run the script
# Documentation: https://robodk.com/doc/en/RoboDK-API.html
# Reference:     https://robodk.com/doc/en/PythonAPI/robodk.html
# Note: It is not required to keep a copy of this file, your Python script is saved with your RDK project

# You can also use the new version of the API:
from robodk import robolink    # RoboDK API
from robodk import robomath    # Robot toolbox
from robodk import time
RDK = robolink.Robolink()


cinta=RDK.Item('CintaUno')
INCREMENTO_MM=50

botella=RDK.Item('Bot')
Posicion1=cinta.Joints().list()


botella.setColor([0.47, 0.27, 0.08, 1])
while Posicion1[0]<2899.0000:
    if cinta.Valid():
        RDK.setParam('Posicion',cinta.Joints())
        cinta.MoveJ(cinta.Joints()+INCREMENTO_MM)
    Posicion1=cinta.Joints().list()

botella.setColor([1.0, 0.55, 0.63, 1])
while Posicion1[0]<4500.0000:
    if cinta.Valid():
        RDK.setParam('Posicion',cinta.Joints())
        cinta.MoveJ(cinta.Joints()+INCREMENTO_MM)
    Posicion1=cinta.Joints().list()

--- Python program AvanzaCinta2 ---
# Type help("robodk.robolink") or help("robodk.robomath") for more information
# Press F5 to run the script
# Documentation: https://robodk.com/doc/en/RoboDK-API.html
# Reference:     https://robodk.com/doc/en/PythonAPI/robodk.html
# Note: It is not required to keep a copy of this file, your Python script is saved with your RDK project

# You can also use the new version of the API:
from robodk import robolink    # RoboDK API
from robodk import robomath    # Robot toolbox
from robodk import time
RDK = robolink.Robolink()


cinta=RDK.Item('CintaSalidas')
INCREMENTO_MM=50


Posicion1=cinta.Joints().list()



while Posicion1[0]<2899.0000:
    if cinta.Valid():
        RDK.setParam('Posicion',cinta.Joints())
        cinta.MoveJ(cinta.Joints()+INCREMENTO_MM)
    Posicion1=cinta.Joints().list()

--- Python program ResetBot ---
from robodk import robolink
from robodk import robomath

RDK = robolink.Robolink()

# VARIABLES INICIALES
PonCero = 0

NUMBOTELLA = int(RDK.getParam('NUMBOTELLA1') or 0)
Eliminadas = 0  # Empezamos desde 0

# BORRAR TODAS LAS BOTELLAS DINÁMICAS
for i in range(NUMBOTELLA+1):
    botella = RDK.Item(f'botella{i}')
    if botella.Valid() and "Save" not in botella.Name():
        botella.Delete()
    Eliminadas += 1
botella = RDK.Item(f'botella{0.0}')
#botella.Delete()

# RESET PARAMS
RDK.setParam('CantBot1', PonCero)
RDK.setParam('NUMBOTELLA1', PonCero)
RDK.setParam('ElimBotellas1', PonCero)
RDK.setParam('repes1', PonCero)
RDK.setParam('Prellena1', PonCero)
RDK.setParam('Detectado1', PonCero)
RDK.setParam('NewPick', PonCero)
RDK.setParam('NewPlace', PonCero)

RDK.setParam('Mesa', 1)
RDK.setParam('MesaE', 1)
RDK.setParam('MesaS', 1)
RDK.setParam('Mesa1', 0)
RDK.setParam('Mesa2', 0)
RDK.setParam('Mesa3', 1)

# RESETEAR CINTA Y FRAME
cinta = RDK.Item('CintaUno')
Move = RDK.Item('Move')

if cinta.Valid():
    cinta.setJoints([50])

if Move.Valid():
    Move.setPose(robomath.transl(0, 0, 0))

# CREAR LA PRIMERA BOTELLA
BotellaBase = RDK.Item('Guardado')
FrameBotella = RDK.Item('FrameBotella')
color_granate_marron = [0.50, 0.12, 0.12, 1.0]

if BotellaBase.Valid() and FrameBotella.Valid():
    BotellaBase.Copy()
    botellaNueva = RDK.Paste(FrameBotella)
    botellaNueva.setName("botella0.0")
    botellaNueva.setVisible(True)
    botellaNueva.setColor(color_granate_marron)

--- program ProgCinta1 (robot CintaUno) ---
  while Detectado1==0
  if Prellena1==0
  while Temperatura == 1
  Pausa 500 ms
  end
  while LotesPendientes == 0
  Pausa 500 ms
  end
  Llamar ProgCintaUno
  end
  if Prellena1!=0
  Pausa 5 ms
  end
  end
  Llamar EMERGENCIA

--- Python program ProgCintaUno ---
# Type help("robodk.robolink") or help("robodk.robomath") for more information
# Press F5 to run the script
# Documentation: https://robodk.com/doc/en/RoboDK-API.html
# Reference: https://robodk.com/doc/en/PythonAPI/robodk.html
# Note: It is not required to keep a copy of this file, your Python script is saved with your RDK project

# You can also use the new version of the API:
# Press F5 to run the script
# Documentation: https://robodk.com/doc/en/RoboDK-API.html
# Reference: https://robodk.com/doc/en/PythonAPI/robodk.html

from robodk import robolink    # RoboDK API
from robodk import robomath    # Robot toolbox

RDK = robolink.Robolink()

INCREMENTO_MM = 150

cinta = RDK.Item('CintaUno')
Botella = RDK.Item('botella0.0')
Guardado = RDK.Item('Guardado')
SisRef = RDK.Item('FrameBotella')
Move = RDK.Item('Move')

repes = RDK.getParam('repes1')

if cinta.Valid():

    NUMBOTELLA = RDK.getParam('NUMBOTELLA1')
    NUMBOTELLA += 1

    pose_actual = Move.Pose()
    nueva_pose = pose_actual

    pose = cinta.Pose()
    x_actual = pose[0, 3]

    if x_actual >= 4200:
        cinta.setJoints([0])
        repes = repes + 1
        Move.setPose(robomath.transl(x_actual * repes, 0, 0))
        RDK.setParam('repes1', repes)

    cinta.MoveJ(cinta.Joints() + INCREMENTO_MM)

    Guardado.Copy()
    GuardadoCopia = RDK.Paste(SisRef)
    GuardadoCopia.setName(f'botella{NUMBOTELLA}')

    CantBot = RDK.getParam('CantBot1')
    CantBot += 1

    GuardadoCopia.setPose(robomath.transl(-INCREMENTO_MM * CantBot, 0, 0))

    # GuardadoCopia.setPose(Botella.Pose() * robomath.transl(-INCREMENTO_MM * CantBot))

    GuardadoCopia.setVisible(True)

    RDK.setParam('CantBot1', CantBot)
    RDK.setParam('NUMBOTELLA1', NUMBOTELLA)
    RDK.RunProgram("CrearBotellaBD")

--- Python program ProgB0 ---
from robodk import robolink
from robodk import robomath

RDK = robolink.Robolink()

Sensor = RDK.Item('B0')

Inicio2 = 0
estadodetectado = 0
cuenta = 0

color_rosa_dalsy = [1.0, 0.75, 0.8, 1.0]

botella = RDK.Item(f'botella{Inicio2}')

while True:

    detectado = 1 if botella.Valid() and Sensor.Collision(botella) else 0

    if detectado != estadodetectado:

        if detectado == 1:
            cuenta += 1

            if cuenta == 3:
                cuenta = 0

                # pintar las 3 últimas botellas
                for i in range(3):
                    pinta = RDK.Item(f'botella{Inicio2 - i}')
                    if pinta.Valid():
                        pinta.setColor(color_rosa_dalsy)
                        estadodetectado = detectado

        # avanzar a la siguiente botella
                if detectado == 0:
                    Inicio2 += 1
                    botella = RDK.Item(f'botella{Inicio2}')
                RDK.RunProgram("LlenarBD")


        else:
            if cuenta < 3:
                RDK.setParam('Prellena1', 0)

        estadodetectado = detectado

        # avanzar a la siguiente botella
        if detectado == 0:
            Inicio2 += 1
            botella = RDK.Item(f'botella{Inicio2}')

    robomath.pause(0.01)

--- Python program ProgB1 ---
from robodk import robolink
from robodk import robomath
import paho.mqtt.client as mqtt

RDK = robolink.Robolink()

# MQTT config
broker = "broker.emqx.io"
port = 1883
user = "giiroB22"
passwd = "UPV2024"
station_status_topic = "giirob/pr2/station/mesa/status/sensorB1"

client = mqtt.Client()
client.username_pw_set(user, passwd)
client.connect(broker, port, 60)

Sensor = RDK.Item('B1')
inicio1 = 0
estadodetectado = 0
cuenta = 0

botella = RDK.Item('botella0')

while True:
    if botella.Valid():
        detectado = 1 if Sensor.Collision(botella) else 0

        if detectado != estadodetectado:

            if detectado == 1:
                RDK.setParam('Detectado1', 1)
                RDK.setParam('Prellena1', 1)
                cuenta += 1

                # 📡 Publicar MQTT
                client.publish(station_status_topic, "sensor_detecta")
                print("[MQTT] sensor_detecta")

            else:
                RDK.setParam('Detectado1', 0)

                # 📡 Publicar MQTT
                client.publish(station_status_topic, "sensor_no_detecta")
                print("[MQTT] sensor_no_detecta")

                inicio1 += 1
                botella = RDK.Item(f'botella{inicio1}')

            estadodetectado = detectado

    else:
        inicio1 += 1
        botella = RDK.Item(f'botella{inicio1}')

    robomath.pause(0.01)

--- Python program ProgB2 ---
from robodk import robolink
from robodk import robomath

RDK = robolink.Robolink()

Sensor = RDK.Item('B2')

Inicio2 = 0
estadodetectado = 0
cuenta = 0

color_rosa_dalsy = [1.0, 0.9, 0.5, 1.0]

botella = RDK.Item(f'botella{Inicio2}')

while True:

    detectado = 1 if botella.Valid() and Sensor.Collision(botella) else 0

    if detectado != estadodetectado:

        if detectado == 1:
            cuenta += 1

            if cuenta == 3:
                cuenta = 0

                for i in range(3):
                    pinta = RDK.Item(f'botella{Inicio2 - i}')
                    if pinta.Valid():
                        pinta.setColor(color_rosa_dalsy)
                        estadodetectado = detectado
                if detectado == 0:
                    Inicio2 += 1
                    botella = RDK.Item(f'botella{Inicio2}')
                RDK.RunProgram("TaponarBD")


        else:
            if cuenta < 3:
                RDK.setParam('Prellena1', 0)

        estadodetectado = detectado

        if detectado == 0:
            Inicio2 += 1
            botella = RDK.Item(f'botella{Inicio2}')

    robomath.pause(0.01)

--- program DalsyPickPlace (robot UR5PickDalsy) ---
  Est. Ref.: Cinta Botellas 1
  Est. herr: RobotiQ 2F-85 Gripper (Open) at (0, 0, 130) mm
  Set Pinza=0
  Establecer velocidad (700.0 mm/s)
  Pausa 500 ms
  while MesaE==0
  end
  MesaE=0
  while Detectado1==0
  MoveJ (DalsyPrepick)
  end
  Llamar EMERGENCIA
  Establecer velocidad (200.0 mm/s)
  MoveL (DalsyPick)
  Set Pinza=1
  Llamar PickDalsy
  Pausa 1.0 s
  MoveL (DalsyPrepick)
  Establecer velocidad (900.0 mm/s)
  MoveJ (DalsyPuntoPaso)
  Prellena1=0
  MoveJ (PuntoDePaso2)
  MoveJ (PrePlace)
  Establecer velocidad (200.0 mm/s)
  MoveL (Place) -> target DalsyPlace
  Llamar PlaceDalsy
  Set Pinza=1
  Llamar BorrarBotella
  Pausa 500 ms
  MoveL (PrePlace)
  Establecer velocidad (800.0 mm/s)
  MoveJ (DalsyPuntoPaso)
  Mesa1=1

--- Python program PickDalsy ---
# Type help("robodk.robolink") or help("robodk.robomath") for more information
# Press F5 to run the script
# Documentation: https://robodk.com/doc/en/RoboDK-API.html
# Reference:     https://robodk.com/doc/en/PythonAPI/robodk.html
# Note: It is not required to keep a copy of this file, your Python script is saved with your RDK project

# You can also use the new version of the API:
from robodk import robolink    # RoboDK API
from robodk import robomath    # Robot toolbox
RDK = robolink.Robolink()

# Forward and backwards compatible use of the RoboDK API:
# Remove these 2 lines to follow python programming guidelines
from robodk import *      # RoboDK API
from robolink import *


RDK = robolink.Robolink()

# === Obtener índice global ===
new_pick = RDK.getParam('NewPick')

# === Obtener botella por índice ===
botella = RDK.Item(f'botella{new_pick}')

# === Obtener robot ===
robot = RDK.Item('GripperPick')  # <-- usa el nombre EXACTO del robot en RoboDK
robot2 = RDK.Item('GripperPickV')
# === Verificación básica ===
if botella.Valid() and robot.Valid():

    # === ATTACH OBJECT (Pick simulado) ===
    robot.DetachAll()
    robot.AttachClosest()

    # === Incrementar índice ===
    new_pick += 1.0
    RDK.setParam('NewPick', new_pick)
    robot.setVisible(False)   # Robot invisible
    robot2.setVisible(True)

--- Python program PlaceDalsy ---
# Type help("robodk.robolink") or help("robodk.robomath") for more information
# Press F5 to run the script
# Documentation: https://robodk.com/doc/en/RoboDK-API.html
# Reference:     https://robodk.com/doc/en/PythonAPI/robodk.html

from robodk import robolink    # RoboDK API
from robodk import robomath    # Robot toolbox
from robodk import *
from robolink import *

RDK = robolink.Robolink()

# === Obtener índice global ===
new_Place = RDK.getParam('NewPlace')

# === Obtener botella por índice ===
botella = RDK.Item(f'botella{int(new_Place)}')

# === Obtener robot ===
robot = RDK.Item('GripperPick')  # <-- usa el nombre EXACTO del robot en RoboDK
robot2 = RDK.Item('GripperPickV')

# === Obtener sistema de coordenadas MesaGiratoria ===
mesa = RDK.Item('SistMesaGiratoria')   # <<< AÑADIDO

# === Verificación básica ===
if botella.Valid() and robot.Valid() and mesa.Valid():
    gripper = RDK.Item('GripperPick')


    # Obtener hijos (objetos cogidos)
    hijos = gripper.Childs()

    if len(hijos) > 0:
        objeto = hijos[0]
        if objeto.Valid():
            objeto.Delete()
    # === Soltar objeto del robot ===
    #robot.DetachAll()

    # === Mantener posición absoluta antes de cambiar parent ===
    #pose_abs = botella.PoseAbs()                     # <<< AÑADIDO

    # === Meter la botella en MesaGiratoria ===

    #botella.setParentStatic(mesa)
    #botella.setParent(mesa)                           # <<< AÑADIDO
    #botella.setPoseAbs(pose_abs)
    #botella.setPose(robomath.transl(0, 0, -9000))                  # <<< AÑADIDO

    # === Incrementar índice ===
    new_Place += 1
    RDK.setParam('NewPlace', new_Place)
    robot2.setVisible(False)   # Robot invisible
    robot.setVisible(True)
    RDK.RunProgram("EmpaquetarBD")

--- Python program BorrarBotella ---
from robodk.robolink import Robolink, ITEM_TYPE_OBJECT

RDK = Robolink()

# Obtener la ventosa
gripper = RDK.Item('GripperPick')


    # Obtener hijos (objetos cogidos)
hijos = gripper.Childs()

if len(hijos) > 0:
    objeto = hijos[0]

    if objeto.Valid():
        objeto.Delete()

--- Python program RobotPickAndPlace ---
from robodk.robolink import *
import time

RDK = Robolink()

robot = RDK.Item('UR5PickDalsy')

if not robot.Valid():
    raise Exception("No se encontró el robot")

robot.setSpeed(700, 100)

while True:

    time.sleep(0.5)

    # Esperar MesaE
    while int(RDK.getParam("MesaE")) == 0:
        time.sleep(0.1)

    RDK.setParam("MesaE", 0)

    # Esperar detección
    DalsyPrepick = RDK.Item("DalsyPrepick")

    while int(RDK.getParam("SensorMqtt")) == 0:
        robot.MoveJ(DalsyPrepick)
        time.sleep(0.1)

    # bajar velocidad
    robot.setSpeed(200, 50)

    # PICK
    robot.MoveL(RDK.Item("DalsyPick"))

    PickDalsy = RDK.Item("PickDalsy")
    PickDalsy.RunProgram()
    PickDalsy.WaitFinished()

    time.sleep(1)

    robot.MoveL(DalsyPrepick)

    # subir velocidad
    robot.setSpeed(700, 100)

    robot.MoveJ(RDK.Item("DalsyPuntoPaso"))

    RDK.setParam("Prellena1", 0)

    robot.MoveJ(RDK.Item("PuntoDePaso2"))
    robot.MoveJ(RDK.Item("PrePlace"))

    robot.setSpeed(200, 50)

    robot.MoveL(RDK.Item("DalsyPlace"))

    PlaceDalsy = RDK.Item("PlaceDalsy")
    PlaceDalsy.RunProgram()
    PlaceDalsy.WaitFinished()

    BorrarBotella = RDK.Item("BorrarBotella")
    BorrarBotella.RunProgram()
    BorrarBotella.WaitFinished()

    time.sleep(0.5)

    robot.MoveL(RDK.Item("PrePlace"))

    robot.setSpeed(700, 100)

    robot.MoveJ(RDK.Item("Target 9"))

    time.sleep(1)

    RDK.setParam("Mesa1", 1)

--- program Prog_cajasSalida (robot UR5 SalidaCjas) ---
  Est. Ref.: UR5BaseSalidaCajas
  Est. herr: VentosaSalida
  while MesaS==0
  Pausa 500 ms
  end
  MesaS=0
  MoveJ (prepick_cajamesa)
  MoveL (pick_cajamesa)
  Pausa 1.0 s
  Adjuntar a VentosaSalida
  MoveL (prepick_cajamesa)
  MoveJ (home)
  Llamar EMERGENCIA
  MoveJ (pre_cajacubo)
  MoveL (dentro_cajacubo)
  Llamar Plantilla
  MoveL (pre_cajacubo)
  MoveJ (preplace_cajacinta)
  MoveL (place_cajacinta)
  Separar de VentosaSalida
  Ejecutar AvanzaCajasSalida
  MoveL (preplace_cajacinta)
  Mesa3=1

--- Python program SensorDetectaCaja ---
from robodk import robolink
import time

RDK = robolink.Robolink()

sensor = RDK.Item('sensorDetectaCajaSalida')

print("Sensor activo. Esperando objetos...")

objeto_detectado = None
estado_anterior = 0

while True:

    # Copia de la lista para evitar problemas internos
    items = list(RDK.ItemList())

    objeto_actual = None

    for item in items:
        try:
            # Validación básica
            if not item.Valid():
                continue

            # Evitar detectar el propio sensor
            if item == sensor:
                continue

            # Solo objetos (no robots, tools, etc.)
            if item.Type() != robolink.ITEM_TYPE_OBJECT:
                continue

            # Solo visibles
            if not item.Visible():
                continue

            # 🔥 Detección de colisión
            if sensor.Collision(item):
                objeto_actual = item
                break

        except:
            # Ignorar cualquier item inválido o corrupto
            continue

    detectado = 1 if objeto_actual is not None else 0

    # Detectar cambio de estado
    if detectado != estado_anterior:

        if detectado == 1:
            objeto_detectado = objeto_actual

            # Mostrar nombre sin romper el script
            try:
                print("Objeto detectado:", objeto_detectado.Name())
            except:
                print("Objeto detectado (nombre no disponible)")

            # Ejecutar programa de RoboDK correctamente
            prog = RDK.Item("Prog_cajasSalida", robolink.ITEM_TYPE_PROGRAM)
            if prog.Valid():
                prog.RunCode()
            else:
                print("⚠ Programa no encontrado o inválido")

        estado_anterior = detectado

    time.sleep(0.01)

--- Python program Plantilla ---
from robodk import robolink    # RoboDK API
from robodk import robomath    # Robot toolbox
RDK = robolink.Robolink()
from robodk.robolink import *
from robodk.robomath import *

caja_para_cerrar = RDK.Item('caja_cerradaPLANTILLA')
herramienta = RDK.Item('VentosaSalida', ITEM_TYPE_TOOL)

caja_para_cerrar.setVisible(False, False)
caja_para_cerrar.setParentStatic(herramienta)
pose_caja_para_cerrar = xyzrpw_2_pose( [ 2.182, 97.233, 6.226, 90.610, -0.743, -89.126 ] )

for obj in herramienta.Childs():
    if obj.Name() != 'caja_cerradaPLANTILLA':
        obj.Delete()
        break #espero que solo haya 1 elemento pillado que sea la caja

caja_para_cerrar.setVisible(False, False)
caja_para_cerrar.setParentStatic(herramienta)
pose_caja_para_cerrar = xyzrpw_2_pose( [ 2.182, 97.233, 6.226, 90.610, -0.743, -89.126 ] )
#[ 2.182, 97.233, 6.226, 90.610, -0.743, -89.126 ]

caja_para_cerrar.setPose(pose_caja_para_cerrar)

caja_para_cerrar.setVisible(True, True)

RDK.Render()

--- Python program AvanzaCajasSalida ---
# Type help("robodk.robolink") or help("robodk.robomath") for more information
# Press F5 to run the script
# Documentation: https://robodk.com/doc/en/RoboDK-API.html
# Reference:     https://robodk.com/doc/en/PythonAPI/robodk.html
# Note: It is not required to keep a copy of this file, your Python script is saved with your RDK project

# You can also use the new version of the API:
from robodk import robolink, robomath
import time

RDK = robolink.Robolink()

frame_cinta = RDK.Item('cinta2')

INCREMENTO_MM = 50
PASOS_MAXIMOS = 33
DELAY = 0.05

print("Cinta en ejecución continua")

# Diccionario para llevar el progreso de cada caja
progreso = {}

while True:
    for caja in frame_cinta.Childs():
        name = caja.Name()

        # Solo cajas cerradas visibles
        if 'caja_cerrada' in name and caja.Visible():

            # Si es la primera vez que vemos esta caja inicializamos sus pasos
            if name not in progreso:
                progreso[name] = 0

            # Si aún no ha llegado al límite de pasos, avanza
            if progreso[name] < PASOS_MAXIMOS:

                pose = caja.Pose()
                pose = pose * robomath.transl(0, INCREMENTO_MM, 0)
                caja.setPose(pose)

                progreso[name] += 1

            else:
                # Cuando llega al límite se oculta
                caja.setVisible(False)
                print(name, "ocultada")

    time.sleep(DELAY)

--- Python program MoverMesa ---
# Type help("robodk.robolink") or help("robodk.robomath") for more information
# Press F5 to run the script
# Documentation: https://robodk.com/doc/en/RoboDK-API.html
# Reference:     https://robodk.com/doc/en/PythonAPI/robodk.html
# Note: It is not required to keep a copy of this file, your Python script is saved with your RDK project

# You can also use the new version of the API:
from robodk import robolink    # RoboDK API
from robodk import robomath
from robodk.robolink import Robolink

# Robot toolbox
RDK = Robolink()
import time

mesa=RDK.Item('MesaGiratoria')
sisRef=RDK.Item('Place_caja')
if mesa.Valid():
    giro=mesa.Joints().list()

if( (giro[0]-90) <  (-200) ):
    giro[0] = 200
    for i in range(0,9):
        giro[0] = giro[0] - 10
        mesa.setJoints(giro)
        time.sleep(0.1)
else:

    for i in range(0,9):
        giro[0] = giro[0]  -10
        mesa.setJoints(giro)
        time.sleep(0.1)


RDK.setParam('Mesa', 1)
RDK.setParam('MesaE', 1)
RDK.setParam('MesaS', 1)
RDK.setParam('Mesa1', 0)
RDK.setParam('Mesa2', 0)
RDK.setParam('Mesa3', 0)

--- program MoverMesaBucle (robot UR5PickDalsy) ---
  if Mesa1==1
  if Mesa2==1
  if Mesa3==1
  Llamar EMERGENCIA
  Llamar MoverMesa
  end
  end
  end

--- program Main (robot UR5PickDalsy) ---
  Llamar ResetBD
  Ejecutar CrearLotesBD
  Llamar ResetBot
  Llamar Inicializar_contador
  Ejecutar ProgB0
  Ejecutar ProgB1
  Ejecutar ProgB2
  Ejecutar ProgCinta1
  Ejecutar RobotPickAndPlace
  Ejecutar Sensor_inicial
  Ejecutar Sensor_place
  Ejecutar Main_sensor
  Ejecutar SensorDetectaCaja
  Ejecutar MoverMesaBucle
  Ejecutar mqttlistenerCinta
  Ejecutar mqttlistenerTEMP
  Ejecutar mqttlistenerDecCaja

--- Python program mqttlistenerCinta ---
#from robodk import robolink    # RoboDK API
#from robodk import robomath    # Robot toolbox
#RDK = robolink.Robolink()

#import paho.mqtt.client as mqtt
#import RobotController as rc

#import paho.mqtt.client as mqtt
#import RobotController as rc

#broker="broker.emqx.io"
#port=1883
#user="giirob222"
#passwd="UPV2024"
#base_topic="giirob/pr2/station/"
#station_name="demo"
#station_commands_topic="giirob/pr2/station/mesa/commands"
#station_status_topic="giirob/pr2/station/mesa/status"

#def on_message(mqttc, obj, msg):
#    payload = msg.payload.decode('utf-8')
#    topic = msg.topic
#    qos = msg.qos
#    rc.handle_message(mqttc, topic, payload)

#mqttc = mqtt.Client(mqtt.CallbackAPIVersion.VERSION2)
#mqttc.on_message = on_message
#mqttc.username_pw_set(username=user, password=passwd)
#mqttc.connect(broker, port, 60)
#mqttc.subscribe(station_commands_topic, 0)
#mqttc.publish(station_status_topic)
#mqttc.loop_forever()

from robodk import robolink
import paho.mqtt.client as mqtt
import RobotControllerCinta as rc  # Importamos nuestro controlador

# Configuración MQTT
broker = "broker.emqx.io"#mqtt.dsic.upv.es/broker.emqx.io
port = 1883
user = "giiroB22"
passwd = "UPV2024"
station_commands_topic = "giirob/pr2/station/mesa/commands/Cinta"
station_status_topic = "giirob/pr2/station/mesa/status"

# Función que se ejecuta al recibir un mensaje
def on_message(client, userdata, msg):
    payload = msg.payload.decode('utf-8')
    topic = msg.topic
    print(f"[MQTT] Recibido: '{payload}' en topic: '{topic}'")
    rc.handle_message(topic, payload)  # solo topic y payload

# Crear cliente MQTT
client = mqtt.Client()
client.username_pw_set(user, passwd)
client.on_message = on_message

# Conectar al broker y suscribirse al topic de comandos
client.connect(broker, port, 60)
client.subscribe(station_commands_topic)

# Publicar status inicial
client.publish(station_status_topic, "online")
print("[MQTT] Publicado status: online")

# Bucle principal
client.loop_forever()

--- Python program RobotControllerCinta ---
from robodk import robolink
RDK = robolink.Robolink()

variables = {
    "SensorMqtt": 0,
    "EMERGENCIA" :0
}

def set_robodk_variable(name, value):
    try:
        RDK.setParam(name, str(value))
        print(f"[RoboDK] {name} = {value}")
    except Exception as e:
        print(f"ERROR: {e}")


def handle_message(topic, payload):

    payload = payload.strip()


    # -------------------------
    # SENSOR MQTT
    # -------------------------
    if payload == "SensorMqtt":
        variables["SensorMqtt"] = 1

    elif payload == "NotSensorMqtt":
        variables["SensorMqtt"] = 0


    # -------------------------
    # EMERGENCIA
    # -------------------------

    elif payload == "EMERGENCIA":
        variables["EMERGENCIA"] = 1

    elif payload == "LIBERADO":
        variables["EMERGENCIA"] = 0

    else:
        print(f"[Controller] No reconocido: {payload}")
        return

    # -------------------------
    # DEBUG
    # -------------------------

    print(f"[Controller] SensorMqtt = {variables['SensorMqtt']}")
    print(f"[Controller] EMERGENCIA = {variables['EMERGENCIA']}")
    # -------------------------
    # UPDATE ROBO DK
    # -------------------------
    set_robodk_variable("SensorMqtt", variables["SensorMqtt"])
    set_robodk_variable("EMERGENCIA", variables["EMERGENCIA"])

--- Python program mqttlistenerTEMP ---
#from robodk import robolink    # RoboDK API
#from robodk import robomath    # Robot toolbox
#RDK = robolink.Robolink()

#import paho.mqtt.client as mqtt
#import RobotController as rc

#import paho.mqtt.client as mqtt
#import RobotController as rc

#broker="broker.emqx.io"
#port=1883
#user="giirob222"
#passwd="UPV2024"
#base_topic="giirob/pr2/station/"
#station_name="demo"
#station_commands_topic="giirob/pr2/station/mesa/commands"
#station_status_topic="giirob/pr2/station/mesa/status"

#def on_message(mqttc, obj, msg):
#    payload = msg.payload.decode('utf-8')
#    topic = msg.topic
#    qos = msg.qos
#    rc.handle_message(mqttc, topic, payload)

#mqttc = mqtt.Client(mqtt.CallbackAPIVersion.VERSION2)
#mqttc.on_message = on_message
#mqttc.username_pw_set(username=user, password=passwd)
#mqttc.connect(broker, port, 60)
#mqttc.subscribe(station_commands_topic, 0)
#mqttc.publish(station_status_topic)
#mqttc.loop_forever()

from robodk import robolink
import paho.mqtt.client as mqtt
import RobotControllerTEMP as rc  # Importamos nuestro controlador

# Configuración MQTT
broker = "broker.emqx.io"#mqtt.dsic.upv.es/broker.emqx.io
port = 1883
user = "giiroB22"
passwd = "UPV2024"
station_commands_topic = "giirob/pr2/station/mesa/commands/TEMP"
station_status_topic = "giirob/pr2/station/mesa/status"

# Función que se ejecuta al recibir un mensaje
def on_message(client, userdata, msg):
    payload = msg.payload.decode('utf-8')
    topic = msg.topic
    print(f"[MQTT] Recibido: '{payload}' en topic: '{topic}'")
    rc.handle_message(topic, payload)  # solo topic y payload

# Crear cliente MQTT
client = mqtt.Client()
client.username_pw_set(user, passwd)
client.on_message = on_message

# Conectar al broker y suscribirse al topic de comandos
client.connect(broker, port, 60)
client.subscribe(station_commands_topic)

# Publicar status inicial
client.publish(station_status_topic, "online")
print("[MQTT] Publicado status: online")

# Bucle principal
client.loop_forever()

--- Python program mqttlistenerDecCaja ---
#from robodk import robolink    # RoboDK API
#from robodk import robomath    # Robot toolbox
#RDK = robolink.Robolink()

#import paho.mqtt.client as mqtt
#import RobotController as rc

#import paho.mqtt.client as mqtt
#import RobotController as rc

#broker="broker.emqx.io"
#port=1883
#user="giirob222"
#passwd="UPV2024"
#base_topic="giirob/pr2/station/"
#station_name="demo"
#station_commands_topic="giirob/pr2/station/mesa/commands"
#station_status_topic="giirob/pr2/station/mesa/status"

#def on_message(mqttc, obj, msg):
#    payload = msg.payload.decode('utf-8')
#    topic = msg.topic
#    qos = msg.qos
#    rc.handle_message(mqttc, topic, payload)

#mqttc = mqtt.Client(mqtt.CallbackAPIVersion.VERSION2)
#mqttc.on_message = on_message
#mqttc.username_pw_set(username=user, password=passwd)
#mqttc.connect(broker, port, 60)
#mqttc.subscribe(station_commands_topic, 0)
#mqttc.publish(station_status_topic)
#mqttc.loop_forever()

from robodk import robolink
import paho.mqtt.client as mqtt
import RobotControllerDecCaja as rc  # Importamos nuestro controlador

# Configuración MQTT
broker = "broker.emqx.io"#mqtt.dsic.upv.es/broker.emqx.io
port = 1883
user = "giiroB22"
passwd = "UPV2024"
station_commands_topic = "giirob/pr2/station/mesa/commands/DecCaja"
station_status_topic = "giirob/pr2/station/mesa/status"

# Función que se ejecuta al recibir un mensaje
def on_message(client, userdata, msg):
    payload = msg.payload.decode('utf-8')
    topic = msg.topic
    print(f"[MQTT] Recibido: '{payload}' en topic: '{topic}'")
    rc.handle_message(topic, payload)  # solo topic y payload

# Crear cliente MQTT
client = mqtt.Client()
client.username_pw_set(user, passwd)
client.on_message = on_message

# Conectar al broker y suscribirse al topic de comandos
client.connect(broker, port, 60)
client.subscribe(station_commands_topic)

# Publicar status inicial
client.publish(station_status_topic, "online")
print("[MQTT] Publicado status: online")

# Bucle principal
client.loop_forever()

--- Python program RobotControllerTEMP ---
from robodk import robolink
RDK = robolink.Robolink()

variables = {
    "Temperatura": 0
}

def set_robodk_variable(name, value):
    try:
        RDK.setParam(name, str(value))
        print(f"[RoboDK] {name} = {value}")
    except Exception as e:
        print(f"ERROR: {e}")


def handle_message(topic, payload):

    payload = payload.strip()

    # -------------------------
    # TEMPERATURA
    # -------------------------
    if payload == "Temperatura_alta":
        variables["Temperatura"] = 1

    elif payload == "Temperatura_correcta":
        variables["Temperatura"] = 0

    else:
        print(f"[Controller] No reconocido: {payload}")
        return

    # -------------------------
    # DEBUG
    # -------------------------
    print(f"[Controller] Temperatura = {variables['Temperatura']}")

    # -------------------------
    # UPDATE ROBO DK
    # -------------------------
    set_robodk_variable("Temperatura", variables["Temperatura"])

--- Python program RobotControllerDecCaja ---
from robodk import robolink
RDK = robolink.Robolink()

variables = {
    "Ini_Detecta_Caja":0
}

def set_robodk_variable(name, value):
    try:
        RDK.setParam(name, str(value))
        print(f"[RoboDK] {name} = {value}")
    except Exception as e:
        print(f"ERROR: {e}")


def handle_message(topic, payload):

    payload = payload.strip()

    # -------------------------
    # TEMPERATURA
    # -------------------------

    if payload == "Detecto_Caja":
        variables["Ini_Detecta_Caja"] = 1

    elif payload == "No_Detecto_Caja":
        variables["Ini_Detecta_Caja"] = 0

    else:
        print(f"[Controller] No reconocido: {payload}")
        return

    # -------------------------
    # DEBUG
    # -------------------------

    print(f"[Controller] Ini_Detecta_Caja = {variables['Ini_Detecta_Caja']}")
    # -------------------------
    # UPDATE ROBO DK
    # -------------------------

    set_robodk_variable("Ini_Detecta_Caja", variables["Ini_Detecta_Caja"])

--- Python program ConsultarBD ---
from robodk.robolink import *
import psycopg2
import time

RDK = Robolink()

conn = psycopg2.connect(
    host="127.0.0.1",
    database="postgres",
    user="postgres",
    password="30082004Aa",
    port="5432"
)

cur = conn.cursor()

print("Sistema iniciado")

while True:
    try:
        cur.execute("""
            SELECT COUNT(*)
            FROM lote
            WHERE estado IN ('pendiente', 'proceso')
        """)

        cantidad = cur.fetchone()[0]

        print("Cantidad:", cantidad)

        if cantidad > 0:
            RDK.setParam('LotesPendientes', '1')
        else:
            RDK.setParam('LotesPendientes', '0')


        RDK.Render()

    except Exception as e:
        print("Error:", e)
        RDK.setParam('LotesPendientes', '0')

    time.sleep(1)

--- Python program CrearBotellaBD ---
import psycopg2

conn = psycopg2.connect(
    host="127.0.0.1",
    database="postgres",
    user="postgres",
    password="30082004Aa",
    port="5432"
)

cur = conn.cursor()

cur.execute("""
    SELECT id
    FROM lote
    WHERE estado IN ('pendiente', 'proceso')
    ORDER BY id
    LIMIT 1
""")

resultado = cur.fetchone()

print("Resultado lote:", resultado)

if resultado:

    lote_id = resultado[0]

    cur.execute("""
        INSERT INTO botellas (
            llenada,
            taponada,
            empaquetada,
            lote_id
        )
        VALUES (FALSE, FALSE, FALSE, %s)
    """, (lote_id,))

    conn.commit()

    print("Botella insertada")

else:
    print("No hay lote disponible")

cur.close()
conn.close()

--- Python program LlenarBD ---
import psycopg2

conn = psycopg2.connect(
    host="127.0.0.1",
    database="postgres",
    user="postgres",
    password="30082004Aa",
    port="5432"
)

cur = conn.cursor()

# 1. Buscar 3 primeras botellas NO llenadas
cur.execute("""
    SELECT codigo
    FROM botellas
    WHERE llenada = FALSE
    ORDER BY codigo
    LIMIT 3
""")

botellas = cur.fetchall()

print("Botellas seleccionadas:", botellas)

# 2. Si hay botellas, marcarlas como llenadas
if len(botellas) > 0:

    for b in botellas:
        cur.execute("""
            UPDATE botellas
            SET llenada = TRUE
            WHERE codigo = %s
        """, (b[0],))

    conn.commit()

    print(" Bloque de llenado ejecutado")

else:
    print(" No hay botellas disponibles")

cur.close()
conn.close()

--- Python program ResetBD ---
import psycopg2

conn = psycopg2.connect(
    host="127.0.0.1",
    database="postgres",
    user="postgres",
    password="30082004Aa",
    port="5432"
)

cur = conn.cursor()

print(" Iniciando RESET completo...")

try:
    # 1. Borrar botellas
    cur.execute("DELETE FROM botellas;")
    print("✔ Botellas eliminadas")

    # 2. Borrar lotes
    cur.execute("DELETE FROM lote;")
    print("✔ Lotes eliminados")

    # 3. Reiniciar IDs (SERIAL)
    cur.execute("ALTER SEQUENCE botellas_codigo_seq RESTART WITH 1;")
    print("✔ Secuencia botellas reiniciada")

    cur.execute("ALTER SEQUENCE lote_id_seq RESTART WITH 1;")
    print("✔ Secuencia lotes reiniciada")

    conn.commit()

    print(" RESET COMPLETO FINALIZADO")

except Exception as e:
    print(" Error durante reset:", e)
    conn.rollback()

finally:
    cur.close()
    conn.close()

--- Python program EmpaquetarBD ---
import psycopg2

conn = psycopg2.connect(
    host="127.0.0.1",
    database="postgres",
    user="postgres",
    password="30082004Aa",
    port="5432"
)

cur = conn.cursor()

print("🔍 Buscando botella para empaquetar...")

try:
    # 1. Buscar primera botella lista para empaquetar
    cur.execute("""
        SELECT codigo
        FROM botellas
        WHERE llenada = TRUE
        AND empaquetada = FALSE
        ORDER BY codigo
        LIMIT 1
    """)

    botella = cur.fetchone()

    if botella:

        codigo = botella[0]

        # 2. Marcar como empaquetada
        cur.execute("""
            UPDATE botellas
            SET empaquetada = TRUE
            WHERE codigo = %s
        """, (codigo,))

        conn.commit()

        print(f"Botella {codigo} empaquetada")

    else:
        print(" No hay botellas listas para empaquetar")

except Exception as e:
    print(" Error:", e)
    conn.rollback()

finally:
    cur.close()
    conn.close()

--- Python program TaponarBD ---
import psycopg2

conn = psycopg2.connect(
    host="127.0.0.1",
    database="postgres",
    user="postgres",
    password="30082004Aa",
    port="5432"
)

cur = conn.cursor()

cur.execute("""
    SELECT codigo
    FROM botellas
    WHERE taponada = FALSE
    ORDER BY codigo
    LIMIT 3
""")

botellas = cur.fetchall()

print("Botellas seleccionadas:", botellas)

if len(botellas) > 0:

    for b in botellas:
        cur.execute("""
            UPDATE botellas
            SET taponada = TRUE
            WHERE codigo = %s
        """, (b[0],))

    conn.commit()

    print("✔ Bloque de taponado ejecutado")

else:
    print("⚠ No hay botellas disponibles")

cur.close()
conn.close()

--- Python program CrearLotesBD ---
import psycopg2

conn = psycopg2.connect(
    host="127.0.0.1",
    database="postgres",
    user="postgres",
    password="30082004Aa",
    port="5432"
)

cur = conn.cursor()

print(" Creando nuevo lote...")

try:
    cur.execute("""
        INSERT INTO lote (estado)
        VALUES ('pendiente')
    """)

    conn.commit()

    print(" Lote creado en estado PENDIENTE")

except Exception as e:
    print(" Error creando lote:", e)
    conn.rollback()

finally:
    cur.close()
    conn.close()

--- Python program TerminarLotesBD ---
import psycopg2
import time

conn = psycopg2.connect(
    host="127.0.0.1",
    database="postgres",
    user="postgres",
    password="30082004Aa",
    port="5432"
)

cur = conn.cursor()

print("Monitor de lotes iniciado...")

while True:
    try:
        # 1. Buscar lote activo
        cur.execute("""
            SELECT id
            FROM lote
            WHERE estado IN ('pendiente', 'proceso')
            ORDER BY id
            LIMIT 1
        """)

        lote = cur.fetchone()

        if lote:

            lote_id = lote[0]

            # 2. Contar empaquetadas del lote
            cur.execute("""
                SELECT COUNT(*)
                FROM botellas
                WHERE empaquetada = TRUE
                AND lote_id = %s
            """, (lote_id,))

            total = cur.fetchone()[0]

            print(f" Lote {lote_id} → {total}/30 empaquetadas")

            # 3. Si llega a 30 → cerrar lote
            if total >= 30:

                cur.execute("""
                    UPDATE lote
                    SET estado = 'terminado'
                    WHERE id = %s
                """, (lote_id,))

                conn.commit()

                print(f" LOTE {lote_id} TERMINADO")

        else:
            print(" No hay lote activo")

    except Exception as e:
        print("Error:", e)
        conn.rollback()

    time.sleep(1)
